FUNCTION_BLOCK FB_SaMElementClearing EXTENDS FB_SaMElement
VAR
END_VAR

METHOD FB_init : BOOL
VAR_INPUT
	bInitRetains : BOOL; // if TRUE, the retain variables are initialized (warm start / cold start)
	bInCopyCode : BOOL;  // if TRUE, the instance afterwards gets moved into the copy code (online change)
END_VAR
THIS^.bTypeActive		:= TRUE;

THIS^.SetText (eLocation := E_BaseLocation.pl, wsDescription := "Czyszczenie");
THIS^.SetText (eLocation := E_BaseLocation.en, wsDescription := "Clearing");
THIS^.SetText (eLocation := E_BaseLocation.de, wsDescription := "Clearing");
THIS^.SetName (stName := THIS^.GetTexts ());
END_METHOD

METHOD public GetNextState : E_BaseMachineState
VAR_INPUT
END_VAR
GetNextState		:= E_BaseMachineState.Stopped;
END_METHOD

METHOD PUBLIC InvokeStateForTopElement : BOOL
VAR_INPUT
	itfTopElement		: ITF_BaseSaMStateMethod;
END_VAR
InvokeStateForTopElement	:= itfTopElement.SP_Clearing ();
END_METHOD

END_FUNCTION_BLOCK

(* stored: Version 1.1.0.1
   POU FB_SaMElementClearing: Id {83b8bb63-7191-0117-2d7d-1f57e6e237b6}, SpecialFunc None
   Method FB_init: Id {7ef8520e-3b5d-0559-01d9-1a6f0bd6c212}
   Method GetNextState: Id {8440fe79-1106-0707-0ebf-6450d74ebe46}
   Method InvokeStateForTopElement: Id {7d9e5f25-6546-0666-33ef-7807e180de33} *)
